Universal Robots PolyScope program: rtde_control_loop.urp

Program rtde_control_loop (createdIn=3.2.19275 lastSavedIn=3.3.19470 directory=/home/rwi/programs installation=default robotSerialNumber=0000200006)
Calibrated DH parameters: a=[0, -0.425, -0.39225, 0, 0, 0]; d=[0.089159, 0, 0, 0.10915, 0.09465, 0.0823]; alpha=[1.570796, 0, 0, 1.570796, -1.570796, 0]; deltaTheta=[0, 0, 0, 0, 0, 0]
BeforeStart
  setp := Joint_6_name
  Script: rtde_set_watchdog("input_int_register_0", 1, "PAUSE")
Robot Program (runOnlyOnce=false motionType=MoveJ speed=1.047198 acceleration=1.396263 recalculateMotions=false)
  Script: write_output_integer_register(0, 0)
  Script: sync()
  MoveL speed 250 mm/s, acceleration 1200 mm/s^2 (recalculateMotions=false) feature=Base
    Waypoint Waypoint (Variable): variable=setp
  Script: write_output_integer_register(0, 1)
  Script: sync()
Thread Thread_1 (runOnlyOnce=false trackProgramExecution=false)
  setp := Joint_6_name
  Loop Forever
    tmp := p[0,0,0,0,0,0]
    Script: tmp[0] = read_input_float_register(0)
    Script: tmp[1] = read_input_float_register(1)
    Script: tmp[2] = read_input_float_register(2)
    Script: tmp[3] = read_input_float_register(3)
    Script: tmp[4] = read_input_float_register(4)
    Script: tmp[5] = read_input_float_register(5)
    If tmp != p[0,0,0,0,0,0]
      setp := tmp
    Script: sync()
